TYPE FB_UdpConnection_cmd :
STRUCT
	//Wird verbinden TRUE verbindet sich der FB auf die angegebene Adresse und Port
	verbinden : BOOL;
	//Den unter text angegebene String senden
	senden : BOOL;
	//Der zu sendende Text
	message : STRING(255);
	//Empfangene Message auslesen
	messageAuslesen : BOOL;
	
	//Die Verbindung trennen
	trennen : BOOL;
	//Verwirft alle noch nicht ausgelesenen Nachtichten
	messagePufferLeeren : BOOL;
	//Fehler quitieren
	reset : BOOL;
END_STRUCT
END_TYPE

(* stored: Version 1.1.0.1, ProductVersion 3.1.4018.5
   DUT FB_UdpConnection_cmd: Id {18412e52-29a5-421c-bfda-0886357b7a75} *)
